(* Logix 5000 project; controller Comas_L4 vendor 1 type 14 code 193 rev 30.11; software revision 30.02; part 12 of 12 *)
(* tags used below, declared in another part *)
   Axe_Codeur_Four : AXIS_CIP_DRIVE;
   CO_Axe_Codeur_Four_Conv_Cons : REAL;
   CO_Top_Once_Axe_Virtuel : BOOL;
   CO_Top_Once_Decoreuse : BOOL;
   CO_Top_Once_Doseuse : BOOL;
   Cpt_Det_Produit : REAL;
   Cpt_Det_Produit2 : REAL;
   Cpt_Fin_Det_Produit : REAL;
   Cpt_Fin_Det_Produit2 : REAL;
   Cpt_Mini_Entre_Produit : REAL;
   Cpt_Mini_Entre_Produit2 : REAL;
   Delta_Avance_Tapis_Four : REAL;
   Det_Produit : BOOL;
   Det_Produit2 : BOOL;
   Distance_CPT_Presence_Produit : DINT;
   Distance_Decoreuse : DINT;
   Distance_Doseuse : DINT;
   ENT_CPT_Synchronisme : ALIAS FOR Local:2:I.Pt06.Data;
   ENT_CPT_Synchronisme2 : ALIAS FOR Local:2:I.Pt05.Data;
   Front_Cpt_Det_PRoduit : FBD_ONESHOT;
   Front_Cpt_Det_PRoduit2 : FBD_ONESHOT;
   Front_Det_produit : FBD_ONESHOT;
   Front_Det_produit2 : FBD_ONESHOT;
   Front_Det_Produit_Filtre : FBD_ONESHOT;
   Front_Det_Produit_Filtre2 : FBD_ONESHOT;
   g_Modulo_Codeur_Four : DINT;
   g_Unwind_Axe_Codeur_Four : DINT;
   Index_Tableau_Tapis : DINT;
   Longueur_Maxi_Tapis_Four : REAL;
   Position_old_Tapis_Four : REAL;
   Position_temp_Tapis_Four : REAL;
   RECETTE_EC : UDT_RECIPE;
   Tableau_Presence_Produit : UDT_REGISTRE_TAPIS[200];
(* Main, continued *)

ROUTINE Registre_Tapis_Entree   (* structured text *)
   // Variable
   Longueur_Maxi_Tapis_Four:=10000;
   Distance_CPT_Presence_Produit:=RECETTE_EC.Comas.Distance_CPT_Presence_Produit;
   Distance_Decoreuse:=RECETTE_EC.Comas.Distance_Decoreuse_mm;
   Distance_Doseuse:=RECETTE_EC.Comas.Distance_Doseuse_mm;
   
   GSV(Axis,Axe_Codeur_Four,PositionUnwind,g_Unwind_Axe_Codeur_Four);
   g_Modulo_Codeur_Four:=(g_Unwind_Axe_Codeur_Four/CO_Axe_Codeur_Four_Conv_Cons);
   
   // Calcul delta avance
   Position_temp_Tapis_Four:=Axe_Codeur_Four.ActualPosition;
   Delta_Avance_Tapis_Four:=Position_temp_Tapis_Four-Position_old_Tapis_Four;
   IF Delta_Avance_Tapis_Four<=-(g_Modulo_Codeur_Four/2) THEN
   	Delta_Avance_Tapis_Four:=Delta_Avance_Tapis_Four+g_Modulo_Codeur_Four;
   END_IF;
   IF Delta_Avance_Tapis_Four>=(g_Modulo_Codeur_Four/2) THEN
   	Delta_Avance_Tapis_Four:=g_Modulo_Codeur_Four-Delta_Avance_Tapis_Four;
   END_IF;
   Position_old_Tapis_Four:=Position_temp_Tapis_Four;
   
   // Tableaux principaux
   FOR Index_Tableau_Tapis:=1 TO 190 BY 1 DO
   	// Tableau Longueur
   	IF (Tableau_Presence_Produit[Index_Tableau_Tapis].Position<Longueur_Maxi_Tapis_Four)
   		THEN
   		Tableau_Presence_Produit[Index_Tableau_Tapis].Position:=Tableau_Presence_Produit[Index_Tableau_Tapis].Position+Delta_Avance_Tapis_Four;
   	ELSE
   		Tableau_Presence_Produit[Index_Tableau_Tapis].Position:=Longueur_Maxi_Tapis_Four;
   	END_IF;
   END_FOR;
   
   // ////////////////////////////////////
   // Controle Longueur Cellule N°1
   // ////////////////////////////////////
   
   // RAZ Data
   IF RECETTE_EC.Comas.Reserve_Real3=0 THEN
   	RECETTE_EC.Comas.Reserve_Real3:=1;
   END_IF;
   IF RECETTE_EC.Comas.Reserve_Real4=0 THEN
   	RECETTE_EC.Comas.Reserve_Real4:=1;
   END_IF;
   IF RECETTE_EC.Comas.Reserve_Real5=0 THEN
   	RECETTE_EC.Comas.Reserve_Real5:=5;
   END_IF;
   
   // ///////////////////////
   // Cellule 1
   // ///////////////////////
   // Detection de Front
   OSRI(Front_Det_produit);
   Front_Det_produit.InputBit:= NOT ENT_CPT_Synchronisme;
   
   // Détection
   IF NOT ENT_CPT_Synchronisme THEN
   	IF Cpt_Det_Produit<50000 THEN
   		Cpt_Det_Produit:=Cpt_Det_Produit+Delta_Avance_Tapis_Four;
   	END_IF;
   ELSE
   	Cpt_Det_Produit:=0;
   END_IF;
   
   Front_Cpt_Det_PRoduit.InputBit:=Cpt_Det_Produit>=RECETTE_EC.Comas.Reserve_Real3;
   OSRI(Front_Cpt_Det_PRoduit);
   
   IF Front_Cpt_Det_PRoduit.OutputBit AND Cpt_Mini_Entre_Produit>=RECETTE_EC.Comas.Reserve_Real5  THEN
   	Det_Produit:=1;
   END_IF;
   
   // Fin Detection
   IF ENT_CPT_Synchronisme THEN
   	IF Cpt_Fin_Det_Produit<50000 THEN
   		Cpt_Fin_Det_Produit:=Cpt_Fin_Det_Produit+Delta_Avance_Tapis_Four;
   	END_IF;
   ELSE
   	Cpt_Fin_Det_Produit:=0;
   END_IF;
   IF Cpt_Fin_Det_Produit>=RECETTE_EC.Comas.Reserve_Real4 THEN
   	Det_Produit:=0;
   END_IF;
   
   Front_Det_Produit_Filtre.InputBit:=Det_Produit;
   OSRI(Front_Det_Produit_Filtre);
   
   // Cpt Mini Entre produit
   IF Front_Det_Produit_Filtre.OutputBit THEN
   	Cpt_Mini_Entre_Produit:=0;
   END_IF;
   IF Cpt_Mini_Entre_Produit<50000 THEN
   	Cpt_Mini_Entre_Produit:=Cpt_Mini_Entre_Produit+Delta_Avance_Tapis_Four;
   END_IF;
   
   
   // ///////////////////////
   // Cellule 2
   // ///////////////////////
   // Detection de Front
   OSRI(Front_Det_produit2);
   Front_Det_produit2.InputBit:= NOT ENT_CPT_Synchronisme2;
   
   // Détection
   IF NOT ENT_CPT_Synchronisme2 THEN
   	IF Cpt_Det_Produit2<50000 THEN
   		Cpt_Det_Produit2:=Cpt_Det_Produit2+Delta_Avance_Tapis_Four;
   	END_IF;
   ELSE
   	Cpt_Det_Produit2:=0;
   END_IF;
   
   Front_Cpt_Det_PRoduit2.InputBit:=Cpt_Det_Produit2>=RECETTE_EC.Comas.Reserve_Real3;
   OSRI(Front_Cpt_Det_PRoduit2);
   
   IF Front_Cpt_Det_PRoduit2.OutputBit AND Cpt_Mini_Entre_Produit2>=RECETTE_EC.Comas.Reserve_Real5  THEN
   	Det_Produit2:=1;
   END_IF;
   
   // Fin Detection
   IF ENT_CPT_Synchronisme2 THEN
   	IF Cpt_Fin_Det_Produit2<50000 THEN
   		Cpt_Fin_Det_Produit2:=Cpt_Fin_Det_Produit2+Delta_Avance_Tapis_Four;
   	END_IF;
   ELSE
   	Cpt_Fin_Det_Produit2:=0;
   END_IF;
   IF Cpt_Fin_Det_Produit2>=RECETTE_EC.Comas.Reserve_Real4 THEN
   	Det_Produit2:=0;
   END_IF;
   
   Front_Det_Produit_Filtre2.InputBit:=Det_Produit2;
   OSRI(Front_Det_Produit_Filtre2);
   
   // Cpt Mini Entre produit
   IF Front_Det_Produit_Filtre2.OutputBit THEN
   	Cpt_Mini_Entre_Produit2:=0;
   END_IF;
   IF Cpt_Mini_Entre_Produit2<50000 THEN
   	Cpt_Mini_Entre_Produit2:=Cpt_Mini_Entre_Produit2+Delta_Avance_Tapis_Four;
   END_IF;
   
   // /////////////////////////////////
   // /////////////////////////////////
   
   IF Front_Det_Produit_Filtre.OutputBit (*Front_Det_produit.OutputBit*) THEN
   	Tableau_Presence_Produit[0].Position:=0;
   	Tableau_Presence_Produit[0].Etat_Produit:=0;
   	// Longueur
   	FOR Index_Tableau_Tapis:=100 TO 1 BY -1 DO
   		Tableau_Presence_Produit[Index_Tableau_Tapis].Position:=Tableau_Presence_Produit[Index_Tableau_Tapis-1].Position;
   		Tableau_Presence_Produit[Index_Tableau_Tapis].Etat_Produit:=Tableau_Presence_Produit[Index_Tableau_Tapis-1].Etat_Produit;
   	END_FOR;
   END_IF;
   
   FOR Index_Tableau_Tapis:=100 TO 1 BY -1 DO
   	IF ((Tableau_Presence_Produit[Index_Tableau_Tapis].Position > (Distance_CPT_Presence_Produit + RECETTE_EC.Comas.Reserve_Real1))
   		AND (Tableau_Presence_Produit[Index_Tableau_Tapis].Position < (Distance_CPT_Presence_Produit + RECETTE_EC.Comas.Pas_Machine))
   		AND NOT Tableau_Presence_Produit[Index_Tableau_Tapis].Etat_Produit.0)
   	THEN
   		Tableau_Presence_Produit[Index_Tableau_Tapis].Etat_Produit.0:=1;
   		CO_Top_Once_Axe_Virtuel:=1;
   	END_IF;
   END_FOR;
   
   FOR Index_Tableau_Tapis:=100 TO 1 BY -1 DO
   	IF ((Tableau_Presence_Produit[Index_Tableau_Tapis].Position > (Distance_Decoreuse + RECETTE_EC.Comas.Reserve_Real2))
   		AND (Tableau_Presence_Produit[Index_Tableau_Tapis].Position < (Distance_Decoreuse + RECETTE_EC.Comas.Pas_Machine))
   		AND NOT Tableau_Presence_Produit[Index_Tableau_Tapis].Etat_Produit.1)
   	THEN
   		Tableau_Presence_Produit[Index_Tableau_Tapis].Etat_Produit.1:=1;
   		CO_Top_Once_Decoreuse:=1;
   	END_IF;
   END_FOR;
   
   FOR Index_Tableau_Tapis:=100 TO 1 BY -1 DO
   	IF ((Tableau_Presence_Produit[Index_Tableau_Tapis].Position > (Distance_Doseuse + RECETTE_EC.Comas.Reserve_Real2))
   		AND (Tableau_Presence_Produit[Index_Tableau_Tapis].Position < (Distance_Doseuse + RECETTE_EC.Comas.Pas_Machine))
   		AND NOT Tableau_Presence_Produit[Index_Tableau_Tapis].Etat_Produit.2)
   	THEN
   		Tableau_Presence_Produit[Index_Tableau_Tapis].Etat_Produit.2:=1;
   		CO_Top_Once_Doseuse:=1;
   	END_IF;
   END_FOR;
   
   
END_ROUTINE
END_PROGRAM
